Staubli VAL3: pickPlate.pgx

public program pickPlate(num nPlate (dimensions=1))
begin
  //robot at pHotel[0] or jHome
  call goHotel(0)
  open(flange)
  movel(appro(pHotel[nPlate],trPickPlateHor),flange,mNomSpeed)
  movel(appro(pHotel[nPlate],trPickPlateVer),flange,mNomSpeed)
  movel(pHotel[nPlate],flange,mNomSpeed)
  close(flange)
  delay(1)
  movel(appro(pHotel[nPlate],trPickPlateVer),flange,mNomSpeed)
  movel(appro(pHotel[nPlate],trPickPlateHor),flange,mNomSpeed)
  movel(pHotel[0],flange,mNomSpeed)
  waitEndMove()
  nHoldingPlate=nPlate
end
